(* Logix 5000 project; controller unittest vendor 1 type 14 code 211 rev 34.11; software revision 34.03 *)
// Indicon LLC
// unittesting plc file

TASK MainTask (continuous, watchdog 500 ms) : MainProgram, CoilWithNoInput, InputWithNoCoil, DuplicatedCoil, NoneFlaggingLogic, LogixOperand
TASK SafetyTask (periodic, rate 20 ms, priority 10, watchdog 20 ms, safety) : SafetyProgram

MODULES
   Local : vendor 1 type 14 code 211 (ICP 0, rev 34.11)
END_MODULES

TYPE za_Parent :
STRUCT
   a : BOOL;
   b : BOOL;
   c : BOOL;
END_STRUCT
END_TYPE

ADD_ON_INSTRUCTION unittest_aoi   (* revision 1.0 *)
// Revision note:
// initial release
VAR_INPUT
   Input : DINT; {required}
END_VAR
VAR_OUTPUT
   Output : DINT; {access Read Only, required}
END_VAR
VAR_IN_OUT
   InOut : DINT; {required}
END_VAR
VAR
   LocalTag : DINT; {access None}
END_VAR

ROUTINE Logic   (* ladder *)
END_ROUTINE
END_ADD_ON_INSTRUCTION

VAR_GLOBAL   (* controller tags *)
   AlwaysOn : BOOL;   // Global Always On
   gCoilWithNoInput : BOOL;   // Global Coil With No Input
   gCoilWithNoInputAlias : BOOL;   // Global Coil With No Input Alias Secondary
   gDuplicatedCoil : BOOL;   // Global Duplicated Coil
   gDuplicatedCoilAlias : BOOL;
   gFirstOperand : BOOL;
   gInputWithNoCoil : BOOL;   // Global Input With No Coil
   gInputWithNoCoilAlias : BOOL;   // Global Input With No Coil Alias
   gSafeBool : BOOL;
   gSafeInteger : DINT;
   gSafeLatch : BOOL;
   gSafeUnlatch : BOOL;
   gStruct : za_Parent;
   MyValue : DINT;
   SecondOperand : DINT;
   SomeStruct : za_Parent;
END_VAR

PROGRAM CoilWithNoInput   (* main routine main *)
VAR
   pCoilWithNoInput : ALIAS FOR gCoilWithNoInputAlias;   // Program Coil With No Input
END_VAR

ROUTINE main   (* ladder *)
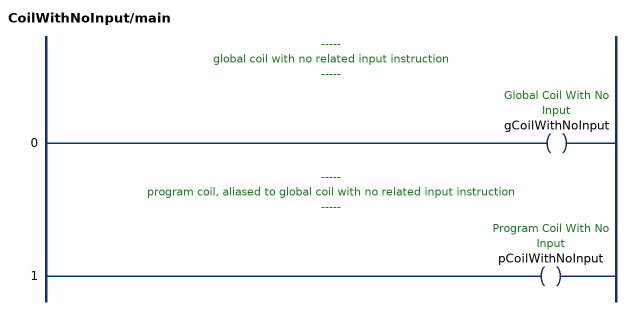
   // -----
   // global coil with no related input instruction
   // -----
   0: OTE(gCoilWithNoInput);
   // -----
   // program coil, aliased to global coil with no related input instruction
   // -----
   1: OTE(pCoilWithNoInput);
END_ROUTINE
END_PROGRAM

PROGRAM DuplicatedCoil   (* main routine main *)
VAR
   pDuplicatedCoil : ALIAS FOR gDuplicatedCoilAlias;
END_VAR

ROUTINE main   (* ladder *)
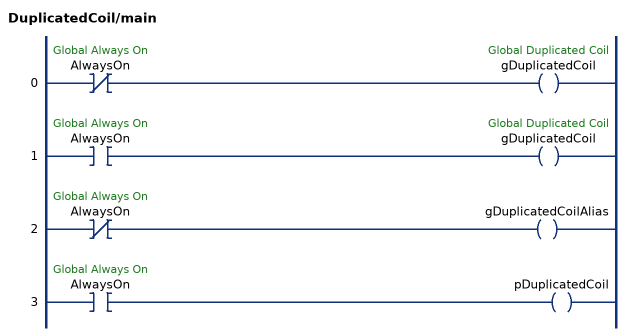
   0: XIO(AlwaysOn)OTE(gDuplicatedCoil);
   1: XIC(AlwaysOn)OTE(gDuplicatedCoil);
   2: XIO(AlwaysOn)OTE(gDuplicatedCoilAlias);
   3: XIC(AlwaysOn)OTE(pDuplicatedCoil);
END_ROUTINE
END_PROGRAM

PROGRAM InputWithNoCoil   (* main routine main *)
VAR
   pInputWithNoCoil : ALIAS FOR gInputWithNoCoilAlias;
END_VAR

ROUTINE main   (* ladder *)
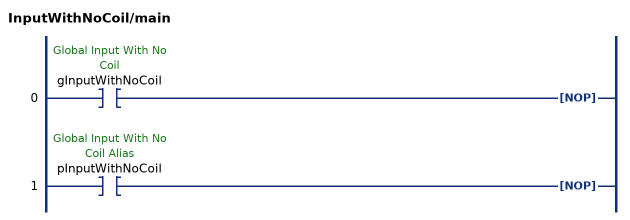
   0: XIC(gInputWithNoCoil)NOP();
   1: XIC(pInputWithNoCoil)NOP();
END_ROUTINE
END_PROGRAM

PROGRAM LogixOperand   (* main routine main *)
VAR
   DeeperAliasing : ALIAS FOR pStruct.c;
   FirstOperand : ALIAS FOR gFirstOperand;   // First Operand In Controller
   LocalProgramTagOnly : BOOL;   // Local Program Tag Only
   pStruct : ALIAS FOR gStruct;
END_VAR

ROUTINE main   (* ladder *)
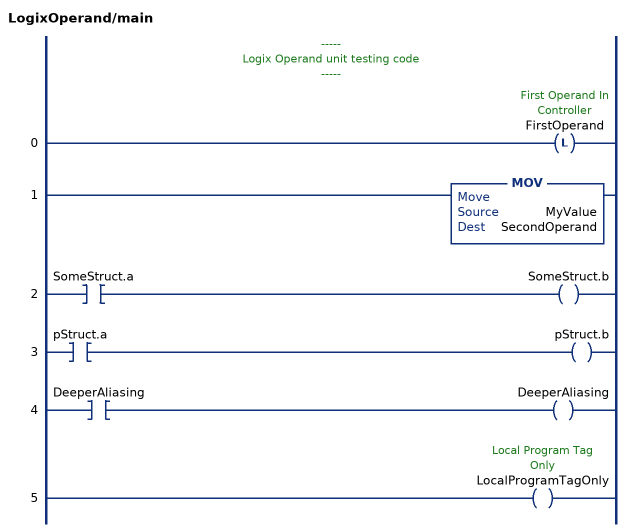
   // -----
   // Logix Operand unit testing code
   // -----
   0: OTL(FirstOperand);
   1: MOV(MyValue,SecondOperand);
   2: XIC(SomeStruct.a)OTE(SomeStruct.b);
   3: XIC(pStruct.a)OTE(pStruct.b);
   4: XIC(DeeperAliasing)OTE(DeeperAliasing);
   5: OTE(LocalProgramTagOnly);
END_ROUTINE
END_PROGRAM

PROGRAM MainProgram   (* main routine main *)

ROUTINE main   (* ladder *)
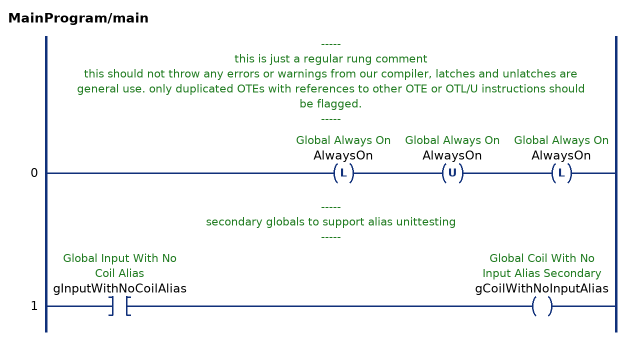
   // -----
   // this is just a regular rung comment
   // this should not throw any errors or warnings from our compiler, latches and unlatches are general use. only duplicated OTEs with references to other OTE or OTL/U instructions should be flagged.
   // -----
   0: OTL(AlwaysOn)OTU(AlwaysOn)OTL(AlwaysOn);
   // -----
   // secondary globals to support alias unittesting
   // -----
   1: XIC(gInputWithNoCoilAlias)OTE(gCoilWithNoInputAlias);
END_ROUTINE
END_PROGRAM

PROGRAM NoneFlaggingLogic   (* main routine main *)

ROUTINE main   (* ladder *)
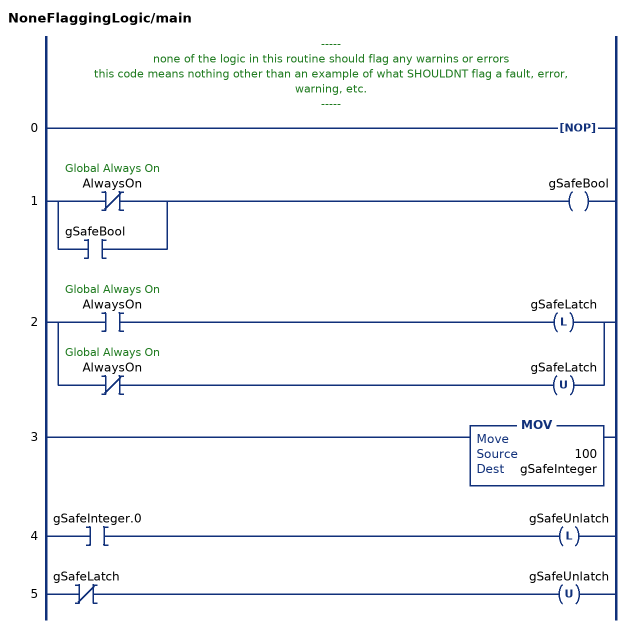
   // -----
   // none of the logic in this routine should flag any warnins or errors
   // this code means nothing other than an example of what SHOULDNT flag a fault, error, warning, etc.
   // -----
   0: NOP();
   1: [XIO(AlwaysOn) ,XIC(gSafeBool) ]OTE(gSafeBool);
   2: [XIC(AlwaysOn) OTL(gSafeLatch) ,XIO(AlwaysOn) OTU(gSafeLatch) ];
   3: MOV(100,gSafeInteger);
   4: XIC(gSafeInteger.0)OTL(gSafeUnlatch);
   5: XIO(gSafeLatch)OTU(gSafeUnlatch);
END_ROUTINE
END_PROGRAM

PROGRAM SafetyProgram   (* main routine MainRoutine, safety *)

ROUTINE MainRoutine   (* ladder *)
   // -----
   // empty routine
   // -----
   0: NOP();
END_ROUTINE
END_PROGRAM
